ABB RobotStudio station: Endelig Levering Station v1.0.rsstn

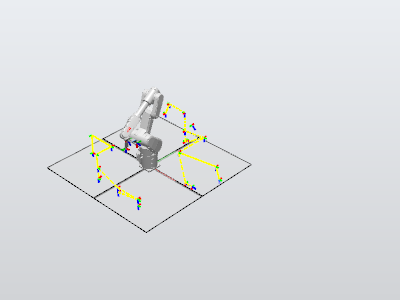
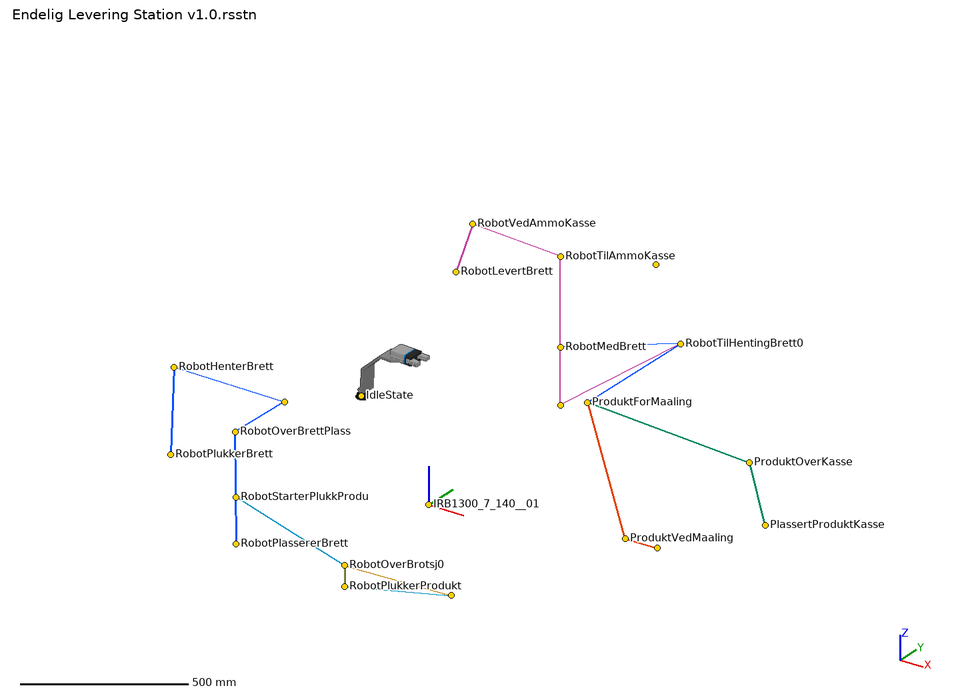
[picture v1: parts stored in the station drawn from their meshes, with robot base, taught points and paths (robot models come from the ABB library and are not in the file)]
Station Station (saved by RobotStudio 23.4.10609.1)
Controller Controller5
  mechanical unit ROB_1: IRB1300_7_140__01, 6 joints, base frame (0, 0, 0) mm
Layout (positions relative to the parent item):
  - IRB1300_7_140__01 [mechanism, from %ABB.RobotStudio.Models.IRB1300%\IRB1300_7_140__01.rslib] at (0, 0, 0) mm; joint values [-1.398, -0.5234, 0.9754, 0.8194, 1.1288, -1.7691] (rad or m)
  - Brakett med sugekopp og griper robot v6 [part] at (144.13, -480.05, 716.42) mm, rotated rx 180 ry 42.11 rz 180 deg, size 302.9 x 67.8 x 90.4 mm
Attachment: Brakett med sugekopp og griper robot v6 is attached to IRB1300_7_140__01 / Link6
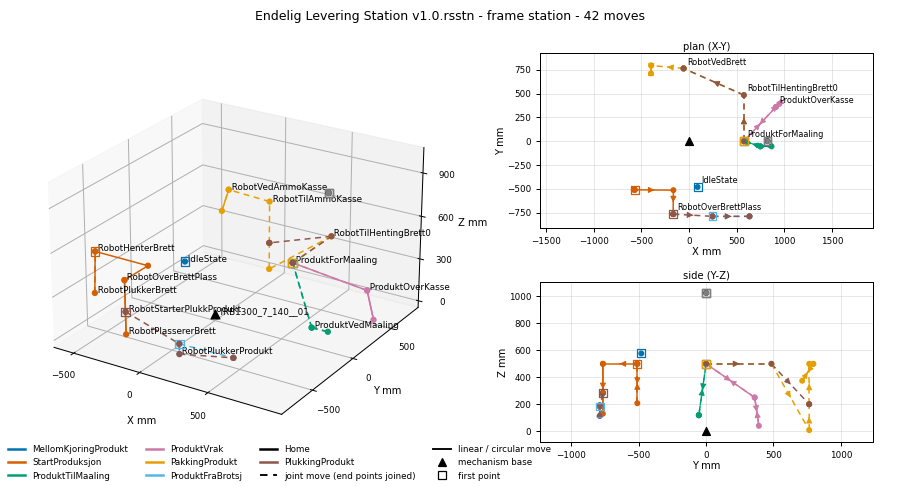
[picture p0: tool path of Endelig Levering Station v1.0.rsstn in frame station, 42 of 46 moves have a stored position in this frame; points joined in program order, loops and branches not executed]
Targets, tools, work objects and paths stored in the station, written as RAPID:
! task T_ROB1
MODULE EndeligLevering
  PERS tooldata TCP_klype:=[TRUE,[[-153.184,0.000002554,86.1346],[0.924787,0,-0.380485,0]],[5,[0,0,0.001],[1,0,0,0],0,0,0]];
  PERS tooldata TCP_Kopp:=[TRUE,[[133.502,0,67.691],[0,0.359227,0,0.93325]],[5,[0,0,0.001],[1,0,0,0],0,0,0]];
  PERS robtarget FraMaalingTilMellomlagring:=[[576.651,0.639056,500],[0.021594,-0.706777,-0.706777,-0.021594],[-1,0,-2,0],[9E+09,9E+09,9E+09,9E+09,9E+09,9E+09]];
  PERS robtarget TilMellomLagring:=[[576.651,485.189,500],[0.021594,-0.706777,-0.706777,-0.021594],[0,0,-2,0],[9E+09,9E+09,9E+09,9E+09,9E+09,9E+09]];
  PERS robtarget VedMellomlagring:=[[-56.7186,765.181,200],[-0.000056241,-0.706749,0.707464,0.000056298],[1,-2,0,1],[9E+09,9E+09,9E+09,9E+09,9E+09,9E+09]];
  PERS robtarget PlassertProdukt:=[[-20.5882,800.001,38],[0.021594,0.706777,-0.706777,0.021594],[1,-2,0,1],[9E+09,9E+09,9E+09,9E+09,9E+09,9E+09]];
  PERS robtarget FerdigLevertProdukt:=[[-56.7186,765.181,200],[-0.000056241,-0.706749,0.707464,0.000056298],[1,-2,0,1],[9E+09,9E+09,9E+09,9E+09,9E+09,9E+09]];
  PERS robtarget IdleState:=[[90.465,-480.047,576.688],[0,1,0,0],[-1,0,-2,0],[9E+09,9E+09,9E+09,9E+09,9E+09,9E+09]];
  PERS robtarget RobotOverBrotsj0:=[[246.805,-788.387,183.38],[0,0.707107,0.707107,0],[-1,0,-2,0],[9E+09,9E+09,9E+09,9E+09,9E+09,9E+09]];
  PERS robtarget RobotPlukkerProdukt:=[[246.805,-788.387,113.38],[0,0.707107,0.707107,0],[-1,0,-2,0],[9E+09,9E+09,9E+09,9E+09,9E+09,9E+09]];
  PERS robtarget RobotOverBrotsj1:=[[246.805,-788.387,183.38],[0,0.707107,0.707107,0],[-1,0,-2,0],[9E+09,9E+09,9E+09,9E+09,9E+09,9E+09]];
  PERS robtarget RobotOverProdukt:=[[635.292,-788.376,191.849],[0,0.707107,0.707107,0],[-1,0,-2,0],[9E+09,9E+09,9E+09,9E+09,9E+09,9E+09]];
  PERS robtarget RobotFyllerBrett:=[[671.53,-827.494,142.55],[0.021594,-0.706777,-0.706777,-0.021594],[-1,0,-2,0],[9E+09,9E+09,9E+09,9E+09,9E+09,9E+09]];
  PERS robtarget RobotOverProdukt0:=[[635.292,-788.376,191.849],[0,0.707107,0.707107,0],[-1,0,-2,0],[9E+09,9E+09,9E+09,9E+09,9E+09,9E+09]];
  PERS robtarget ProduktTilVrak:=[[576.651,0.639056,500],[0.021594,-0.706777,-0.706777,-0.021594],[-1,-2,-1,1],[9E+09,9E+09,9E+09,9E+09,9E+09,9E+09]];
  PERS robtarget ProduktOverKasse:=[[913.152,361.021,250],[0,0.707107,0.707107,0],[0,-2,0,1],[9E+09,9E+09,9E+09,9E+09,9E+09,9E+09]];
  PERS robtarget PlassertProduktKasse:=[[947.915,392.209,40],[0.021594,-0.706777,-0.706777,-0.021594],[0,-2,0,1],[9E+09,9E+09,9E+09,9E+09,9E+09,9E+09]];
  PERS robtarget RobotOverKasse:=[[913.152,361.021,250],[0,0.707107,0.707107,0],[0,-2,0,1],[9E+09,9E+09,9E+09,9E+09,9E+09,9E+09]];
  PERS robtarget RobotFerdigLevertProduktVrak:=[[576.651,0.639056,500],[0.021594,-0.706777,-0.706777,-0.021594],[-1,-2,0,1],[9E+09,9E+09,9E+09,9E+09,9E+09,9E+09]];
  PERS robtarget ProduktKlarTilMaaling:=[[671.53,-827.494,250],[0.021594,-0.706777,-0.706777,-0.021594],[-1,-2,-1,1],[9E+09,9E+09,9E+09,9E+09,9E+09,9E+09]];
  PERS robtarget PlukkerProdukt:=[[671.53,-827.494,142.55],[0.021594,-0.706777,-0.706777,-0.021594],[-1,-2,0,1],[9E+09,9E+09,9E+09,9E+09,9E+09,9E+09]];
  PERS robtarget ProduktForMaaling:=[[576.651,0.639056,500],[0.021594,-0.706777,-0.706777,-0.021594],[-1,-2,0,1],[9E+09,9E+09,9E+09,9E+09,9E+09,9E+09]];
  PERS robtarget ProduktVedMaaling:=[[750.492,-53.2362,118.133],[0.688355,0,0.725374,0],[-1,-1,1,1],[9E+09,9E+09,9E+09,9E+09,9E+09,9E+09]];
  PERS robtarget ProduktMaaling:=[[866.89,-53.2362,119.852],[0.688341,-0.0044336,0.725356,0.00507842],[-1,-1,1,1],[9E+09,9E+09,9E+09,9E+09,9E+09,9E+09]];
  PERS robtarget ProduktVedMaaling0:=[[750.492,-53.2362,118.133],[0.688355,0,0.725374,0],[-1,-1,1,1],[9E+09,9E+09,9E+09,9E+09,9E+09,9E+09]];
  PERS robtarget ProduktForMaaling0:=[[576.651,0.639056,500],[0.021594,-0.706777,-0.706777,-0.021594],[-1,-2,0,1],[9E+09,9E+09,9E+09,9E+09,9E+09,9E+09]];
  PERS robtarget RobotStarterPlukkProdukt:=[[-163.812,-764.841,285],[0,0.707107,0.707107,0],[-2,-3,-5,1],[9E+09,9E+09,9E+09,9E+09,9E+09,9E+09]];
  PERS robtarget ProduktPlukk:=[[-126.381,-803.735,150],[0.021594,-0.706777,-0.706777,-0.021594],[-2,-3,-5,1],[9E+09,9E+09,9E+09,9E+09,9E+09,9E+09]];
  PERS robtarget ProduktPlukk0:=[[-163.812,-764.841,285],[0,0.707107,0.707107,0],[-2,-3,-5,1],[9E+09,9E+09,9E+09,9E+09,9E+09,9E+09]];
  PERS robtarget ProduktOverBrotsj:=[[246.805,-788.387,183.38],[0,0.707107,0.707107,0],[-1,-2,-4,1],[9E+09,9E+09,9E+09,9E+09,9E+09,9E+09]];
  PERS robtarget ProduktPlassertBrotsj:=[[246.805,-788.387,113.38],[0,0.707107,0.707107,0],[-1,-2,-4,1],[9E+09,9E+09,9E+09,9E+09,9E+09,9E+09]];
  PERS robtarget RobotOverBrotsj:=[[246.805,-788.387,183.38],[0,0.707107,0.707107,0],[-1,-2,-4,1],[9E+09,9E+09,9E+09,9E+09,9E+09,9E+09]];
  PERS robtarget RobotHenterBrett:=[[-568.349,-509.47,500],[0,0.999048,0,-0.0436194],[-2,-1,-1,0],[9E+09,9E+09,9E+09,9E+09,9E+09,9E+09]];
  PERS robtarget RobotPlukkerBrett:=[[-580.172,-509.47,207.601],[0,0.999048,0,-0.0436194],[-2,0,0,0],[9E+09,9E+09,9E+09,9E+09,9E+09,9E+09]];
  PERS robtarget RobotFlytterBrett:=[[-568.349,-509.47,500],[0,0.999048,0,-0.0436194],[-2,0,0,0],[9E+09,9E+09,9E+09,9E+09,9E+09,9E+09]];
  PERS robtarget MellomPosisjon:=[[-163.812,-513.339,500],[0,0.707107,0.707107,0],[-2,-1,-1,0],[9E+09,9E+09,9E+09,9E+09,9E+09,9E+09]];
  PERS robtarget RobotOverBrettPlass:=[[-166.881,-764.83,500],[-0.000403746,0.707107,0.707107,-0.000403746],[-2,-1,-1,0],[9E+09,9E+09,9E+09,9E+09,9E+09,9E+09]];
  PERS robtarget RobotPlassererBrett:=[[-163.812,-764.841,130],[0,0.707107,0.707107,0],[-2,-1,-1,0],[9E+09,9E+09,9E+09,9E+09,9E+09,9E+09]];
  PERS robtarget RobotFerdigPlassertBrett:=[[-166.881,-764.83,500],[-0.000403746,0.707107,0.707107,-0.000403746],[-2,-1,-1,0],[9E+09,9E+09,9E+09,9E+09,9E+09,9E+09]];
  PERS robtarget RobotTilHentingBrett:=[[576.651,0.639056,500],[0.021594,-0.706777,-0.706777,-0.021594],[-1,0,0,0],[9E+09,9E+09,9E+09,9E+09,9E+09,9E+09]];
  PERS robtarget RobotTilHentingBrett0:=[[576.651,485.189,500],[0.021594,-0.706777,-0.706777,-0.021594],[0,0,0,0],[9E+09,9E+09,9E+09,9E+09,9E+09,9E+09]];
  PERS robtarget RobotVedBrett:=[[-56.6764,765.183,8],[0,-0.706747,0.707466,0],[1,0,0,0],[9E+09,9E+09,9E+09,9E+09,9E+09,9E+09]];
  PERS robtarget RobotMedBrett:=[[-56.7186,765.181,200],[0.0216655,0.706417,-0.707136,0.0215224],[1,0,0,0],[9E+09,9E+09,9E+09,9E+09,9E+09,9E+09]];
  PERS robtarget RobotTilAmmoKasse:=[[-56.7186,765.181,500],[0.0216655,0.706417,-0.707136,0.0215224],[1,0,0,0],[9E+09,9E+09,9E+09,9E+09,9E+09,9E+09]];
  PERS robtarget RobotVedAmmoKasse:=[[-396.648,795.613,500],[0,-0.706747,0.707466,0],[1,0,0,0],[9E+09,9E+09,9E+09,9E+09,9E+09,9E+09]];
  PERS robtarget RobotLevertBrett:=[[-399.443,713.363,374.009],[0,-0.706747,0.707466,0],[1,0,0,0],[9E+09,9E+09,9E+09,9E+09,9E+09,9E+09]];
  PERS robtarget RobotFerdigLevertBrett:=[[-396.648,795.613,500],[0,-0.706747,0.707466,0],[1,0,0,0],[9E+09,9E+09,9E+09,9E+09,9E+09,9E+09]];
  PERS robtarget HomePosisjon:=[[824.79,1.67817,1025.5],[0.000412889,0.913919,0.000929666,0.405895],[0,-2,2,1],[9E+09,9E+09,9E+09,9E+09,9E+09,9E+09]];
  PERS robtarget HomePos:=[[824.79,1.67817,1025.5],[0.000412889,0.913919,0.000929666,0.405895],[0,-3,2,1],[9E+09,9E+09,9E+09,9E+09,9E+09,9E+09]];
  PROC Main()
    Home;
    StartProduksjon;
    MellomKjoringProdukt;
    WaitDI di2,1;
    PlukkingProdukt;
    WaitTime 1;
    MellomKjoringProdukt;
    WaitDI di4,1;
    PakkingProdukt;
    Home;
  ENDPROC
  PROC MellomKjoringProdukt()
    MoveJ IdleState,vmax,fine,TCP_Kopp\WObj:=wobj0;
    WaitTime 2;
  ENDPROC
  PROC StartProduksjon()
    WaitDI di1,1;
    MoveJ RobotHenterBrett,vmax,fine,TCP_klype\WObj:=wobj0;
    WaitTime 2;
    MoveL RobotPlukkerBrett,v2500,fine,TCP_klype\WObj:=wobj0;
    SetDO do2,1;
    WaitTime 2;
    MoveJ RobotFlytterBrett,vmax,fine,TCP_klype\WObj:=wobj0;
    MoveL MellomPosisjon,v2500,fine,TCP_klype\WObj:=wobj0;
    MoveL RobotOverBrettPlass,v2500,fine,TCP_klype\WObj:=wobj0;
    WaitTime 1;
    MoveL RobotPlassererBrett,v2500,fine,TCP_klype\WObj:=wobj0;
    SetDO do2,0;
    WaitTime 2;
    MoveL RobotFerdigPlassertBrett,v2500,fine,TCP_klype\WObj:=wobj0;
  ENDPROC
  PROC ProduktTilMaaling()
    MoveJ ProduktForMaaling,vmax,fine,TCP_Kopp\WObj:=wobj0;
    MoveJ ProduktVedMaaling,vmax,fine,TCP_Kopp\WObj:=wobj0;
    MoveJ ProduktMaaling,v2500,fine,TCP_Kopp\WObj:=wobj0;
    WaitTime 3;
    MoveJ ProduktVedMaaling0,vmax,fine,TCP_Kopp\WObj:=wobj0;
    MoveJ ProduktForMaaling0,vmax,fine,TCP_Kopp\WObj:=wobj0;
  ENDPROC
  PROC ProduktVrak()
    MoveJ ProduktTilVrak,vmax,fine,TCP_Kopp\WObj:=wobj0;
    MoveL ProduktOverKasse,v2500,fine,TCP_Kopp\WObj:=wobj0;
    MoveL PlassertProduktKasse,v2500,fine,TCP_Kopp\WObj:=wobj0;
    WaitTime 1;
    SetDO do1,0;
    MoveL RobotOverKasse,v2500,fine,TCP_Kopp\WObj:=wobj0;
    MoveJ RobotFerdigLevertProduktVrak,vmax,fine,TCP_Kopp\WObj:=wobj0;
  ENDPROC
  PROC PakkingProdukt()
    MoveJ RobotTilHentingBrett,vmax,fine,TCP_klype\WObj:=wobj0;
    MoveJ RobotTilHentingBrett0,vmax,fine,TCP_klype\WObj:=wobj0;
    MoveJ RobotVedBrett,vmax,fine,TCP_klype\WObj:=wobj0;
    SetDO do2,1;
    WaitTime 1;
    MoveJ RobotMedBrett,v2500,fine,TCP_klype\WObj:=wobj0;
    MoveJ RobotTilAmmoKasse,vmax,fine,TCP_klype\WObj:=wobj0;
    MoveJ RobotVedAmmoKasse,vmax,fine,TCP_klype\WObj:=wobj0;
    MoveL RobotLevertBrett,v2500,fine,TCP_klype\WObj:=wobj0;
    SetDO do2,0;
    WaitTime 1;
    MoveJ RobotFerdigLevertBrett,vmax,fine,TCP_klype\WObj:=wobj0;
  ENDPROC
  PROC ProduktFraBrotsj()
    MoveJ RobotOverBrotsj0,vmax,fine,TCP_Kopp\WObj:=wobj0;
    MoveJ RobotPlukkerProdukt,vmax,fine,TCP_Kopp\WObj:=wobj0;
    SetDO do1,1;
    WaitTime 1;
    MoveL RobotOverBrotsj1,v2500,fine,TCP_Kopp\WObj:=wobj0;
    MoveJ RobotOverProdukt,v2500,fine,TCP_Kopp\WObj:=wobj0;
    WaitTime 1;
  ENDPROC
  PROC Home()
    MoveJ HomePos,v2500,fine,TCP_Kopp\WObj:=wobj0;
    WaitTime 3;
    WaitTime 0.5;
  ENDPROC
  PROC PlukkingProdukt()
    MoveJ RobotStarterPlukkProdukt,vmax,fine,TCP_Kopp\WObj:=wobj0;
    SetDO do1,1;
    MoveJ Offs(ProduktPlukk, x* (-30),y* 30,0),vmax,fine,TCP_Kopp\WObj:=wobj0;
    MoveJ RobotStarterPlukkProdukt,vmax,fine,TCP_Kopp\WObj:=wobj0;
    MoveJ ProduktOverBrotsj,vmax,fine,TCP_Kopp\WObj:=wobj0;
    MoveJ ProduktPlassertBrotsj,vmax,fine,TCP_Kopp\WObj:=wobj0;
    SetDO do1,0;
    WaitTime 3;
    MellomKjoringProdukt;
    WaitDI di3,1;
    WaitTime 3;
    ProduktFraBrotsj;
    MoveJ RobotOverProdukt,v2500,fine,TCP_Kopp\WObj:=wobj0;
    MoveJ Offs(RobotFyllerBrett, x* (-30),y* 30,0),vmax,fine,TCP_Kopp\WObj:=wobj0;
    MellomKjoringProdukt;
    MoveJ RobotOverProdukt,v2500,fine,TCP_Kopp\WObj:=wobj0;
    MoveJ Offs(RobotFyllerBrett, x* (-30),y* 30,0),vmax,fine,TCP_Kopp\WObj:=wobj0;
    ProduktTilMaaling;
    ProduktVrak;
    MoveJ FraMaalingTilMellomlagring,vmax,fine,TCP_Kopp\WObj:=wobj0;
    MoveJ TilMellomLagring,v2500,fine,TCP_Kopp\WObj:=wobj0;
    MoveJ VedMellomlagring,v2500,fine,TCP_Kopp\WObj:=wobj0;
    MoveL Offs(PlassertProdukt,x *(-30),y *30,0),v2500,fine,TCP_Kopp\WObj:=wobj0;
    WaitTime 1;
    SetDO do1,0;
    WaitTime 1;
    MoveL FerdigLevertProdukt,v2500,fine,TCP_Kopp\WObj:=wobj0;
  ENDPROC
  PROC Service()
    MoveJ HomePos,v2500,fine,TCP_Kopp\WObj:=wobj0;
    WaitTime 1;
  ENDPROC
  PROC StartSyklus()
    Main;
    Service;
    WaitTime 30;
  ENDPROC
ENDMODULE

